{attribute 'linkalways'} 
{attribute 'no_explicit_call' := 'This FB is a CLASS and must be accessed using methods or properties'}
{attribute 'enable_dynamic_creation'}
FUNCTION_BLOCK FINAL LT_LREAL EXTENDS Node
VAR
	in1 : _LREAL(0.0);
	in2 : _LREAL(0.0);
	out : _BOOL(FALSE);
END_VAR

METHOD PUBLIC Clone : I_Node
VAR
	pNode : POINTER TO LT_LREAL;
END_VAR
pNode := __NEW(LT_LREAL);
Clone := pNode^;
END_METHOD

METHOD FB_init : BOOL
VAR_INPUT
	bInitRetains : BOOL; // if TRUE, the retain variables are initialized (warm start / cold start)
	bInCopyCode : BOOL;  // if TRUE, the instance afterwards gets moved into the copy code (online change)
END_VAR
AddInput('in1',THIS^.in1);
AddInput('in2',THIS^.in2);
AddOutput('out', THIS^.out);
END_METHOD

METHOD PROTECTED OnExecute
VAR
END_VAR
out.Value := in1.Value < in2.Value;
END_METHOD

END_FUNCTION_BLOCK

(* stored: Version 1.1.0.1, ProductVersion 3.1.4024.15
   POU LT_LREAL: Id {01e8dd0b-6751-4438-a558-e62e7030cf4a}, SpecialFunc None
   Folder Constructor: Id {9c0d37b1-868d-49bf-ae87-0e7436b1602b}
   Method Clone: Id {3a947f0b-3fb2-43fa-b72a-8a8295019640}
   Method FB_init: Id {893fa793-e0f6-416c-a89b-7ecd1badb57c}
   Method OnExecute: Id {b87bd9f1-62e4-4ef6-b2bb-14b34e7bf2dd} *)
